// TIA Portal V18 export
FUNCTION "Recirculation Sequences" : Void   // FC12, LAD
{ S7_Optimized_Access := 'TRUE' }
VERSION : 0.1
// stored: AutoNumber true, IsIECCheckEnabled false, SetENOAutomatically false, UDAEnableTagReadback false
   VAR_TEMP   // added for the SCL form of the ladder/FBD networks
      _w1 : Bool;
   END_VAR
BEGIN

REGION Network 1: A selection
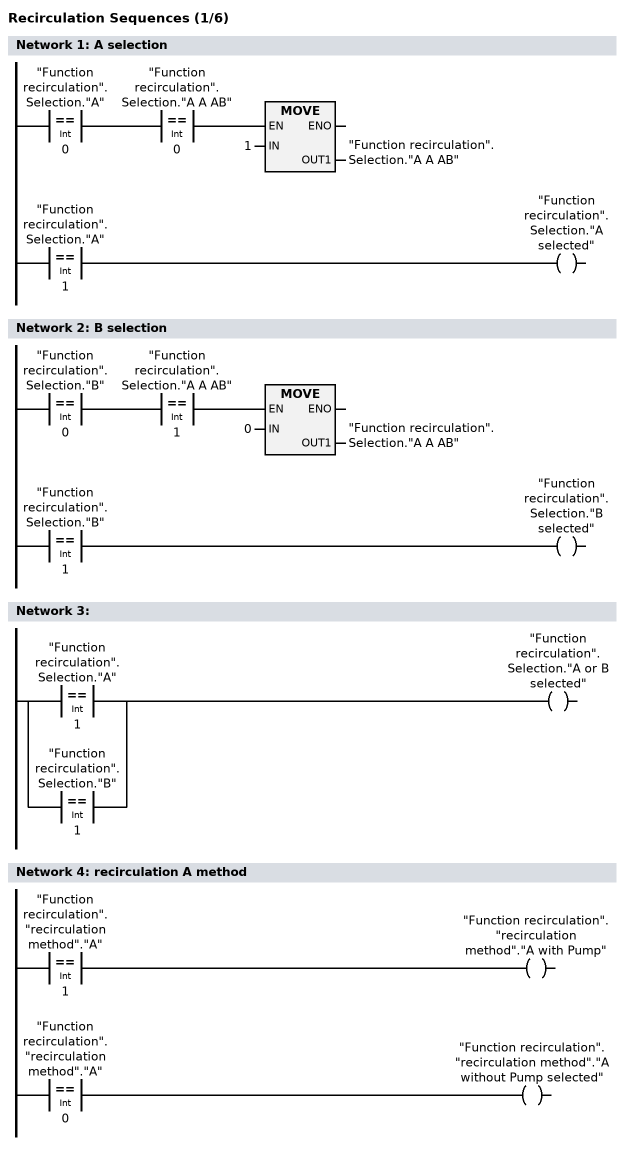
   RUNG wire#powerrail
      { S7_Templates := "SrcType := Int" } EQ_Contact(in1 := "Function recirculation".Selection."A", in2 := 0)
      { S7_Templates := "SrcType := Int" } EQ_Contact(in1 := "Function recirculation".Selection."A A AB", in2 := 0)
      Move(in := 1, out1 => "Function recirculation".Selection."A A AB")
   END_RUNG
   RUNG wire#powerrail
      { S7_Templates := "SrcType := Int" } EQ_Contact(in1 := "Function recirculation".Selection."A", in2 := 1)
      Coil( "Function recirculation".Selection."A selected" )
   END_RUNG
   // the same network as SCL:
   IF ("Function recirculation".Selection."A" = 0) AND ("Function recirculation".Selection."A A AB" = 0) THEN
       "Function recirculation".Selection."A A AB" := 1;
   END_IF;
   "Function recirculation".Selection."A selected" := "Function recirculation".Selection."A" = 1;
END_REGION

REGION Network 2: B selection
   RUNG wire#powerrail
      { S7_Templates := "SrcType := Int" } EQ_Contact(in1 := "Function recirculation".Selection."B", in2 := 0)
      { S7_Templates := "SrcType := Int" } EQ_Contact(in1 := "Function recirculation".Selection."A A AB", in2 := 1)
      Move(in := 0, out1 => "Function recirculation".Selection."A A AB")
   END_RUNG
   RUNG wire#powerrail
      { S7_Templates := "SrcType := Int" } EQ_Contact(in1 := "Function recirculation".Selection."B", in2 := 1)
      Coil( "Function recirculation".Selection."B selected" )
   END_RUNG
   // the same network as SCL:
   IF ("Function recirculation".Selection."B" = 0) AND ("Function recirculation".Selection."A A AB" = 1) THEN
       "Function recirculation".Selection."A A AB" := 0;
   END_IF;
   "Function recirculation".Selection."B selected" := "Function recirculation".Selection."B" = 1;
END_REGION

REGION Network 3
   RUNG wire#powerrail
      { S7_Templates := "SrcType := Int" } EQ_Contact(in1 := "Function recirculation".Selection."A", in2 := 1)
      wire#w1
      Coil( "Function recirculation".Selection."A or B selected" )
   END_RUNG
   RUNG wire#powerrail
      { S7_Templates := "SrcType := Int" } EQ_Contact(in1 := "Function recirculation".Selection."B", in2 := 1)
   END_RUNG wire#w1
   // the same network as SCL:
   "Function recirculation".Selection."A or B selected" := ("Function recirculation".Selection."A" = 1) OR ("Function recirculation".Selection."B" = 1);
END_REGION

REGION Network 4: recirculation A method
   RUNG wire#powerrail
      { S7_Templates := "SrcType := Int" } EQ_Contact(in1 := "Function recirculation"."recirculation method"."A", in2 := 1)
      Coil( "Function recirculation"."recirculation method"."A with Pump" )
   END_RUNG
   RUNG wire#powerrail
      { S7_Templates := "SrcType := Int" } EQ_Contact(in1 := "Function recirculation"."recirculation method"."A", in2 := 0)
      Coil( "Function recirculation"."recirculation method"."A without Pump selected" )
   END_RUNG
   // the same network as SCL:
   "Function recirculation"."recirculation method"."A with Pump" := "Function recirculation"."recirculation method"."A" = 1;
   "Function recirculation"."recirculation method"."A without Pump selected" := "Function recirculation"."recirculation method"."A" = 0;
END_REGION

REGION Network 5: recirculation B method
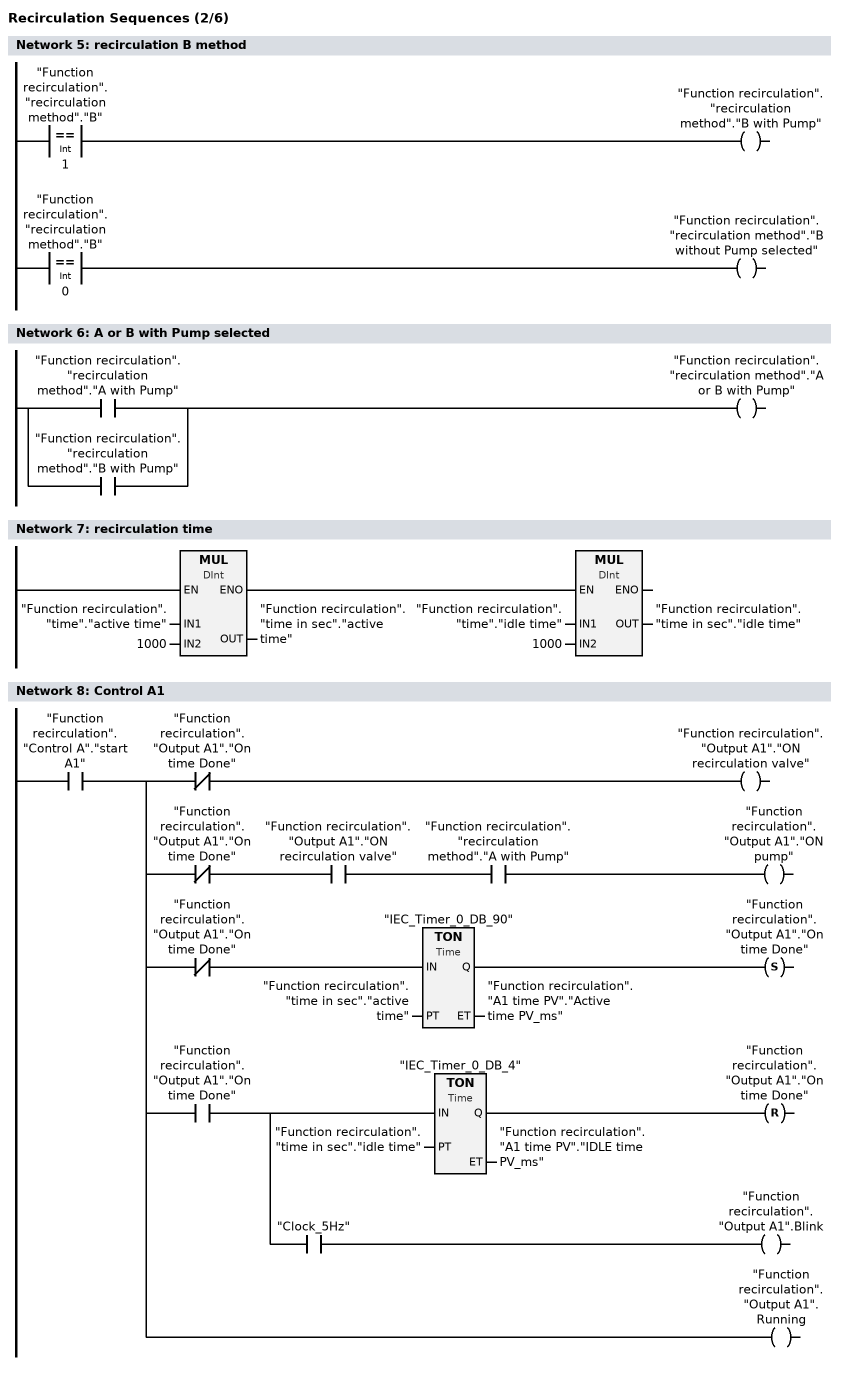
   RUNG wire#powerrail
      { S7_Templates := "SrcType := Int" } EQ_Contact(in1 := "Function recirculation"."recirculation method"."B", in2 := 1)
      Coil( "Function recirculation"."recirculation method"."B with Pump" )
   END_RUNG
   RUNG wire#powerrail
      { S7_Templates := "SrcType := Int" } EQ_Contact(in1 := "Function recirculation"."recirculation method"."B", in2 := 0)
      Coil( "Function recirculation"."recirculation method"."B without Pump selected" )
   END_RUNG
   // the same network as SCL:
   "Function recirculation"."recirculation method"."B with Pump" := "Function recirculation"."recirculation method"."B" = 1;
   "Function recirculation"."recirculation method"."B without Pump selected" := "Function recirculation"."recirculation method"."B" = 0;
END_REGION

REGION Network 6: A or B with Pump selected
   RUNG wire#powerrail
      Contact( "Function recirculation"."recirculation method"."A with Pump" )
      wire#w1
      Coil( "Function recirculation"."recirculation method"."A or B with Pump" )
   END_RUNG
   RUNG wire#powerrail
      Contact( "Function recirculation"."recirculation method"."B with Pump" )
   END_RUNG wire#w1
   // the same network as SCL:
   "Function recirculation"."recirculation method"."A or B with Pump" := "Function recirculation"."recirculation method"."A with Pump" OR "Function recirculation"."recirculation method"."B with Pump";
END_REGION

REGION Network 7: recirculation time
   RUNG wire#powerrail
      { S7_Templates := "SrcType := DInt" } Mul(in1 := "Function recirculation"."time"."active time", in2 := 1000, out => "Function recirculation"."time in sec"."active time")
      { S7_Templates := "SrcType := DInt" } Mul(in1 := "Function recirculation"."time"."idle time", in2 := 1000, out => "Function recirculation"."time in sec"."idle time")
   END_RUNG
   // the same network as SCL:
   "Function recirculation"."time in sec"."active time" := "Function recirculation"."time"."active time" * 1000;
   "Function recirculation"."time in sec"."idle time" := "Function recirculation"."time"."idle time" * 1000;
END_REGION

REGION Network 8: Control A1
   RUNG wire#powerrail
      Contact( "Function recirculation"."Control A"."start A1" )
      wire#w1
      I_Contact( "Function recirculation"."Output A1"."On time Done" )
      Coil( "Function recirculation"."Output A1"."ON recirculation valve" )
   END_RUNG
   RUNG wire#w1
      I_Contact( "Function recirculation"."Output A1"."On time Done" )
      Contact( "Function recirculation"."Output A1"."ON recirculation valve" )
      Contact( "Function recirculation"."recirculation method"."A with Pump" )
      Coil( "Function recirculation"."Output A1"."ON pump" )
   END_RUNG
   RUNG wire#w1
      I_Contact( "Function recirculation"."Output A1"."On time Done" )
      { S7_Templates := "time_type := Time" } "IEC_Timer_0_DB_90".TON(pt := "Function recirculation"."time in sec"."active time", et => "Function recirculation"."A1 time PV"."Active time PV_ms")
      S_Coil( "Function recirculation"."Output A1"."On time Done" )
   END_RUNG
   RUNG wire#w1
      Contact( "Function recirculation"."Output A1"."On time Done" )
      wire#w2
      { S7_Templates := "time_type := Time" } "IEC_Timer_0_DB_4".TON(pt := "Function recirculation"."time in sec"."idle time", et => "Function recirculation"."A1 time PV"."IDLE time PV_ms")
      R_Coil( "Function recirculation"."Output A1"."On time Done" )
   END_RUNG
   RUNG wire#w2
      Contact( "Clock_5Hz" )
      Coil( "Function recirculation"."Output A1".Blink )
   END_RUNG
   RUNG wire#w1
      Coil( "Function recirculation"."Output A1".Running )
   END_RUNG
   // the same network as SCL:
   "Function recirculation"."Output A1"."ON recirculation valve" := "Function recirculation"."Control A"."start A1" AND NOT "Function recirculation"."Output A1"."On time Done";
   "Function recirculation"."Output A1"."ON pump" := "Function recirculation"."Control A"."start A1" AND NOT "Function recirculation"."Output A1"."On time Done" AND "Function recirculation"."Output A1"."ON recirculation valve" AND "Function recirculation"."recirculation method"."A with Pump";
   "IEC_Timer_0_DB_90".TON(IN := "Function recirculation"."Control A"."start A1" AND NOT "Function recirculation"."Output A1"."On time Done",
                           PT := "Function recirculation"."time in sec"."active time",
                           ET => "Function recirculation"."A1 time PV"."Active time PV_ms");
   IF "IEC_Timer_0_DB_90".Q THEN "Function recirculation"."Output A1"."On time Done" := TRUE; END_IF;
   #_w1 := "Function recirculation"."Control A"."start A1" AND "Function recirculation"."Output A1"."On time Done";
   "IEC_Timer_0_DB_4".TON(IN := #_w1,
                          PT := "Function recirculation"."time in sec"."idle time",
                          ET => "Function recirculation"."A1 time PV"."IDLE time PV_ms");
   IF "IEC_Timer_0_DB_4".Q THEN "Function recirculation"."Output A1"."On time Done" := FALSE; END_IF;
   "Function recirculation"."Output A1".Blink := #_w1 AND "Clock_5Hz";
   "Function recirculation"."Output A1".Running := "Function recirculation"."Control A"."start A1";
END_REGION

REGION Network 9: Control A2
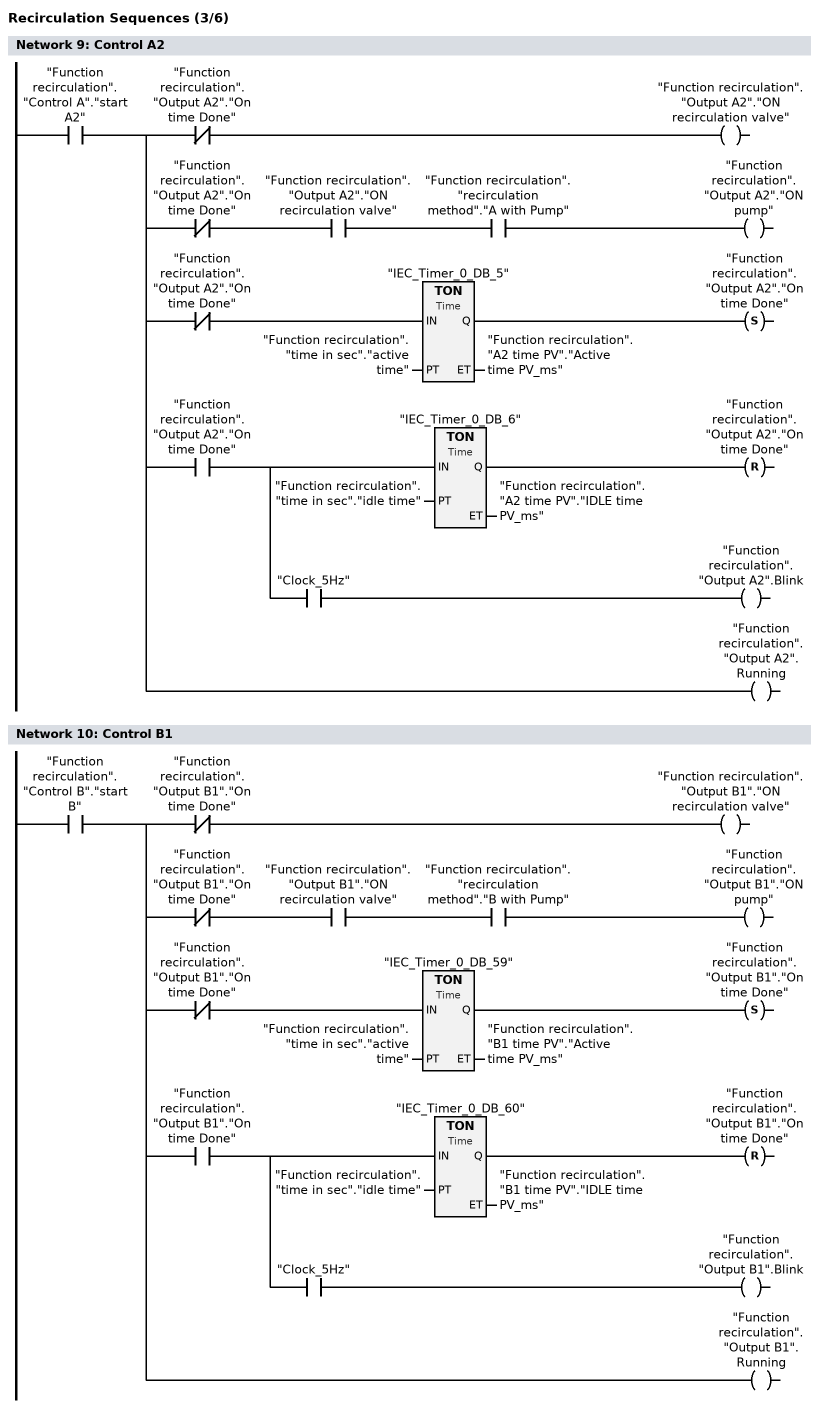
   RUNG wire#powerrail
      Contact( "Function recirculation"."Control A"."start A2" )
      wire#w1
      I_Contact( "Function recirculation"."Output A2"."On time Done" )
      Coil( "Function recirculation"."Output A2"."ON recirculation valve" )
   END_RUNG
   RUNG wire#w1
      I_Contact( "Function recirculation"."Output A2"."On time Done" )
      Contact( "Function recirculation"."Output A2"."ON recirculation valve" )
      Contact( "Function recirculation"."recirculation method"."A with Pump" )
      Coil( "Function recirculation"."Output A2"."ON pump" )
   END_RUNG
   RUNG wire#w1
      I_Contact( "Function recirculation"."Output A2"."On time Done" )
      { S7_Templates := "time_type := Time" } "IEC_Timer_0_DB_5".TON(pt := "Function recirculation"."time in sec"."active time", et => "Function recirculation"."A2 time PV"."Active time PV_ms")
      S_Coil( "Function recirculation"."Output A2"."On time Done" )
   END_RUNG
   RUNG wire#w1
      Contact( "Function recirculation"."Output A2"."On time Done" )
      wire#w2
      { S7_Templates := "time_type := Time" } "IEC_Timer_0_DB_6".TON(pt := "Function recirculation"."time in sec"."idle time", et => "Function recirculation"."A2 time PV"."IDLE time PV_ms")
      R_Coil( "Function recirculation"."Output A2"."On time Done" )
   END_RUNG
   RUNG wire#w2
      Contact( "Clock_5Hz" )
      Coil( "Function recirculation"."Output A2".Blink )
   END_RUNG
   RUNG wire#w1
      Coil( "Function recirculation"."Output A2".Running )
   END_RUNG
   // the same network as SCL:
   "Function recirculation"."Output A2"."ON recirculation valve" := "Function recirculation"."Control A"."start A2" AND NOT "Function recirculation"."Output A2"."On time Done";
   "Function recirculation"."Output A2"."ON pump" := "Function recirculation"."Control A"."start A2" AND NOT "Function recirculation"."Output A2"."On time Done" AND "Function recirculation"."Output A2"."ON recirculation valve" AND "Function recirculation"."recirculation method"."A with Pump";
   "IEC_Timer_0_DB_5".TON(IN := "Function recirculation"."Control A"."start A2" AND NOT "Function recirculation"."Output A2"."On time Done",
                          PT := "Function recirculation"."time in sec"."active time",
                          ET => "Function recirculation"."A2 time PV"."Active time PV_ms");
   IF "IEC_Timer_0_DB_5".Q THEN "Function recirculation"."Output A2"."On time Done" := TRUE; END_IF;
   #_w1 := "Function recirculation"."Control A"."start A2" AND "Function recirculation"."Output A2"."On time Done";
   "IEC_Timer_0_DB_6".TON(IN := #_w1,
                          PT := "Function recirculation"."time in sec"."idle time",
                          ET => "Function recirculation"."A2 time PV"."IDLE time PV_ms");
   IF "IEC_Timer_0_DB_6".Q THEN "Function recirculation"."Output A2"."On time Done" := FALSE; END_IF;
   "Function recirculation"."Output A2".Blink := #_w1 AND "Clock_5Hz";
   "Function recirculation"."Output A2".Running := "Function recirculation"."Control A"."start A2";
END_REGION

REGION Network 10: Control B1
   RUNG wire#powerrail
      Contact( "Function recirculation"."Control B"."start B" )
      wire#w1
      I_Contact( "Function recirculation"."Output B1"."On time Done" )
      Coil( "Function recirculation"."Output B1"."ON recirculation valve" )
   END_RUNG
   RUNG wire#w1
      I_Contact( "Function recirculation"."Output B1"."On time Done" )
      Contact( "Function recirculation"."Output B1"."ON recirculation valve" )
      Contact( "Function recirculation"."recirculation method"."B with Pump" )
      Coil( "Function recirculation"."Output B1"."ON pump" )
   END_RUNG
   RUNG wire#w1
      I_Contact( "Function recirculation"."Output B1"."On time Done" )
      { S7_Templates := "time_type := Time" } "IEC_Timer_0_DB_59".TON(pt := "Function recirculation"."time in sec"."active time", et => "Function recirculation"."B1 time PV"."Active time PV_ms")
      S_Coil( "Function recirculation"."Output B1"."On time Done" )
   END_RUNG
   RUNG wire#w1
      Contact( "Function recirculation"."Output B1"."On time Done" )
      wire#w2
      { S7_Templates := "time_type := Time" } "IEC_Timer_0_DB_60".TON(pt := "Function recirculation"."time in sec"."idle time", et => "Function recirculation"."B1 time PV"."IDLE time PV_ms")
      R_Coil( "Function recirculation"."Output B1"."On time Done" )
   END_RUNG
   RUNG wire#w2
      Contact( "Clock_5Hz" )
      Coil( "Function recirculation"."Output B1".Blink )
   END_RUNG
   RUNG wire#w1
      Coil( "Function recirculation"."Output B1".Running )
   END_RUNG
   // the same network as SCL:
   "Function recirculation"."Output B1"."ON recirculation valve" := "Function recirculation"."Control B"."start B" AND NOT "Function recirculation"."Output B1"."On time Done";
   "Function recirculation"."Output B1"."ON pump" := "Function recirculation"."Control B"."start B" AND NOT "Function recirculation"."Output B1"."On time Done" AND "Function recirculation"."Output B1"."ON recirculation valve" AND "Function recirculation"."recirculation method"."B with Pump";
   "IEC_Timer_0_DB_59".TON(IN := "Function recirculation"."Control B"."start B" AND NOT "Function recirculation"."Output B1"."On time Done",
                           PT := "Function recirculation"."time in sec"."active time",
                           ET => "Function recirculation"."B1 time PV"."Active time PV_ms");
   IF "IEC_Timer_0_DB_59".Q THEN "Function recirculation"."Output B1"."On time Done" := TRUE; END_IF;
   #_w1 := "Function recirculation"."Control B"."start B" AND "Function recirculation"."Output B1"."On time Done";
   "IEC_Timer_0_DB_60".TON(IN := #_w1,
                           PT := "Function recirculation"."time in sec"."idle time",
                           ET => "Function recirculation"."B1 time PV"."IDLE time PV_ms");
   IF "IEC_Timer_0_DB_60".Q THEN "Function recirculation"."Output B1"."On time Done" := FALSE; END_IF;
   "Function recirculation"."Output B1".Blink := #_w1 AND "Clock_5Hz";
   "Function recirculation"."Output B1".Running := "Function recirculation"."Control B"."start B";
END_REGION

REGION Network 11: Recirculation A Active time PV
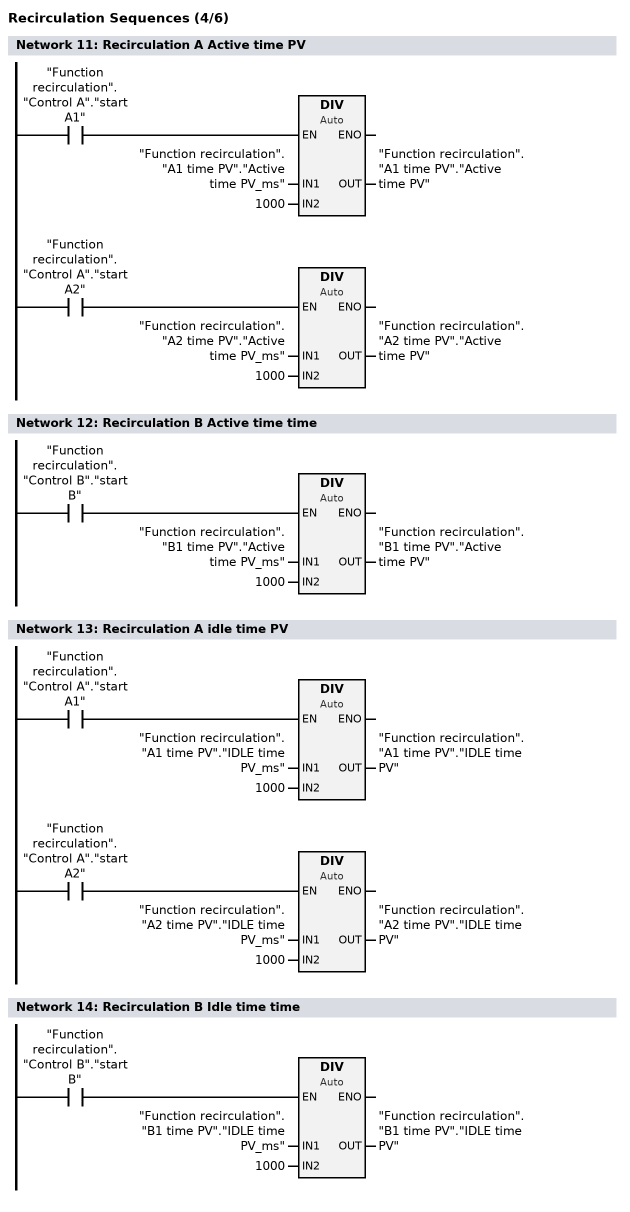
   RUNG wire#powerrail
      Contact( "Function recirculation"."Control A"."start A1" )
      Div(in1 := "Function recirculation"."A1 time PV"."Active time PV_ms", in2 := 1000, out => "Function recirculation"."A1 time PV"."Active time PV")
   END_RUNG
   RUNG wire#powerrail
      Contact( "Function recirculation"."Control A"."start A2" )
      Div(in1 := "Function recirculation"."A2 time PV"."Active time PV_ms", in2 := 1000, out => "Function recirculation"."A2 time PV"."Active time PV")
   END_RUNG
   // the same network as SCL:
   IF "Function recirculation"."Control A"."start A1" THEN
       "Function recirculation"."A1 time PV"."Active time PV" := "Function recirculation"."A1 time PV"."Active time PV_ms" / 1000;
   END_IF;
   IF "Function recirculation"."Control A"."start A2" THEN
       "Function recirculation"."A2 time PV"."Active time PV" := "Function recirculation"."A2 time PV"."Active time PV_ms" / 1000;
   END_IF;
END_REGION

REGION Network 12: Recirculation B Active time time
   RUNG wire#powerrail
      Contact( "Function recirculation"."Control B"."start B" )
      Div(in1 := "Function recirculation"."B1 time PV"."Active time PV_ms", in2 := 1000, out => "Function recirculation"."B1 time PV"."Active time PV")
   END_RUNG
   // the same network as SCL:
   IF "Function recirculation"."Control B"."start B" THEN
       "Function recirculation"."B1 time PV"."Active time PV" := "Function recirculation"."B1 time PV"."Active time PV_ms" / 1000;
   END_IF;
END_REGION

REGION Network 13: Recirculation A idle time PV
   RUNG wire#powerrail
      Contact( "Function recirculation"."Control A"."start A1" )
      Div(in1 := "Function recirculation"."A1 time PV"."IDLE time PV_ms", in2 := 1000, out => "Function recirculation"."A1 time PV"."IDLE time PV")
   END_RUNG
   RUNG wire#powerrail
      Contact( "Function recirculation"."Control A"."start A2" )
      Div(in1 := "Function recirculation"."A2 time PV"."IDLE time PV_ms", in2 := 1000, out => "Function recirculation"."A2 time PV"."IDLE time PV")
   END_RUNG
   // the same network as SCL:
   IF "Function recirculation"."Control A"."start A1" THEN
       "Function recirculation"."A1 time PV"."IDLE time PV" := "Function recirculation"."A1 time PV"."IDLE time PV_ms" / 1000;
   END_IF;
   IF "Function recirculation"."Control A"."start A2" THEN
       "Function recirculation"."A2 time PV"."IDLE time PV" := "Function recirculation"."A2 time PV"."IDLE time PV_ms" / 1000;
   END_IF;
END_REGION

REGION Network 14: Recirculation B Idle time time
   RUNG wire#powerrail
      Contact( "Function recirculation"."Control B"."start B" )
      Div(in1 := "Function recirculation"."B1 time PV"."IDLE time PV_ms", in2 := 1000, out => "Function recirculation"."B1 time PV"."IDLE time PV")
   END_RUNG
   // the same network as SCL:
   IF "Function recirculation"."Control B"."start B" THEN
       "Function recirculation"."B1 time PV"."IDLE time PV" := "Function recirculation"."B1 time PV"."IDLE time PV_ms" / 1000;
   END_IF;
END_REGION

REGION Network 15: A1 Active time to HMI
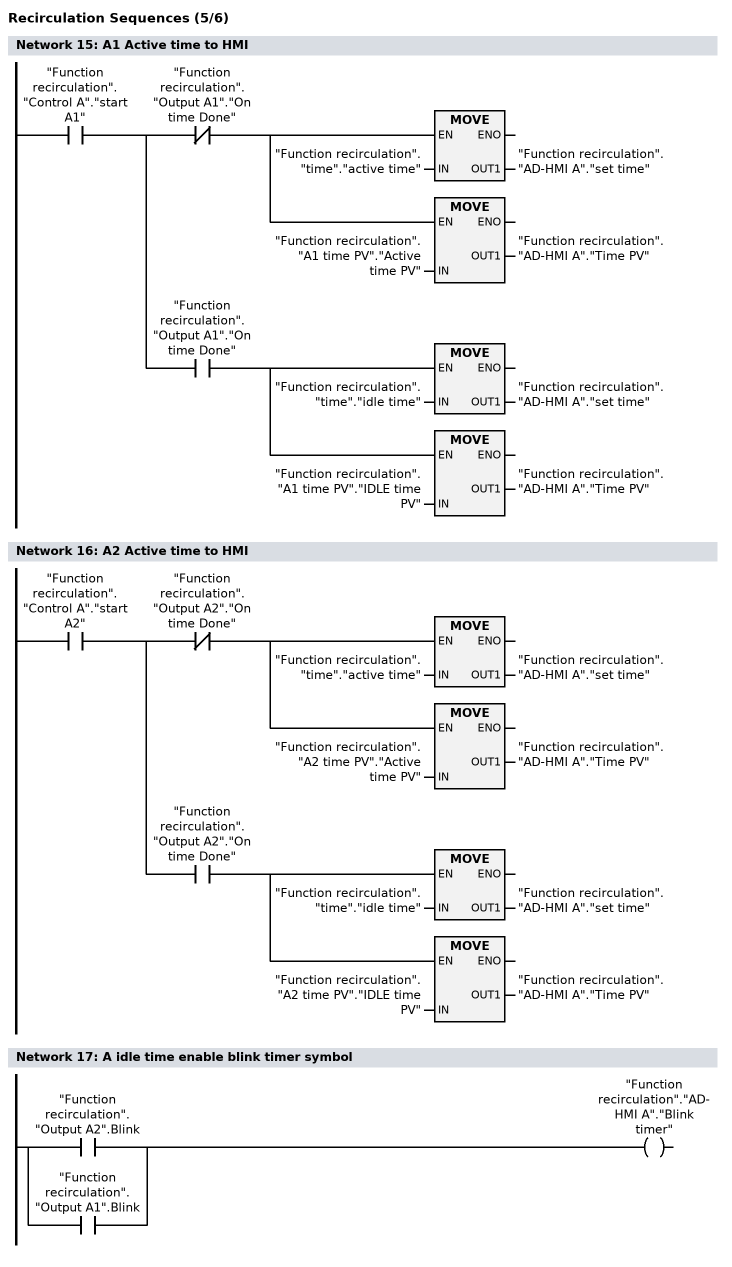
   RUNG wire#powerrail
      Contact( "Function recirculation"."Control A"."start A1" )
      wire#w1
      I_Contact( "Function recirculation"."Output A1"."On time Done" )
      wire#w2
      Move(in := "Function recirculation"."time"."active time", out1 => "Function recirculation"."AD-HMI A"."set time")
   END_RUNG
   RUNG wire#w2
      Move(in := "Function recirculation"."A1 time PV"."Active time PV", out1 => "Function recirculation"."AD-HMI A"."Time PV")
   END_RUNG
   RUNG wire#w1
      Contact( "Function recirculation"."Output A1"."On time Done" )
      wire#w3
      Move(in := "Function recirculation"."time"."idle time", out1 => "Function recirculation"."AD-HMI A"."set time")
   END_RUNG
   RUNG wire#w3
      Move(in := "Function recirculation"."A1 time PV"."IDLE time PV", out1 => "Function recirculation"."AD-HMI A"."Time PV")
   END_RUNG
   // the same network as SCL:
   IF "Function recirculation"."Control A"."start A1" AND NOT "Function recirculation"."Output A1"."On time Done" THEN
       "Function recirculation"."AD-HMI A"."set time" := "Function recirculation"."time"."active time";
       "Function recirculation"."AD-HMI A"."Time PV" := "Function recirculation"."A1 time PV"."Active time PV";
   END_IF;
   IF "Function recirculation"."Control A"."start A1" AND "Function recirculation"."Output A1"."On time Done" THEN
       "Function recirculation"."AD-HMI A"."set time" := "Function recirculation"."time"."idle time";
       "Function recirculation"."AD-HMI A"."Time PV" := "Function recirculation"."A1 time PV"."IDLE time PV";
   END_IF;
END_REGION

REGION Network 16: A2 Active time to HMI
   RUNG wire#powerrail
      Contact( "Function recirculation"."Control A"."start A2" )
      wire#w1
      I_Contact( "Function recirculation"."Output A2"."On time Done" )
      wire#w2
      Move(in := "Function recirculation"."time"."active time", out1 => "Function recirculation"."AD-HMI A"."set time")
   END_RUNG
   RUNG wire#w2
      Move(in := "Function recirculation"."A2 time PV"."Active time PV", out1 => "Function recirculation"."AD-HMI A"."Time PV")
   END_RUNG
   RUNG wire#w1
      Contact( "Function recirculation"."Output A2"."On time Done" )
      wire#w3
      Move(in := "Function recirculation"."time"."idle time", out1 => "Function recirculation"."AD-HMI A"."set time")
   END_RUNG
   RUNG wire#w3
      Move(in := "Function recirculation"."A2 time PV"."IDLE time PV", out1 => "Function recirculation"."AD-HMI A"."Time PV")
   END_RUNG
   // the same network as SCL:
   IF "Function recirculation"."Control A"."start A2" AND NOT "Function recirculation"."Output A2"."On time Done" THEN
       "Function recirculation"."AD-HMI A"."set time" := "Function recirculation"."time"."active time";
       "Function recirculation"."AD-HMI A"."Time PV" := "Function recirculation"."A2 time PV"."Active time PV";
   END_IF;
   IF "Function recirculation"."Control A"."start A2" AND "Function recirculation"."Output A2"."On time Done" THEN
       "Function recirculation"."AD-HMI A"."set time" := "Function recirculation"."time"."idle time";
       "Function recirculation"."AD-HMI A"."Time PV" := "Function recirculation"."A2 time PV"."IDLE time PV";
   END_IF;
END_REGION

REGION Network 17: A idle time enable blink timer symbol
   RUNG wire#powerrail
      Contact( "Function recirculation"."Output A2".Blink )
      wire#w1
      Coil( "Function recirculation"."AD-HMI A"."Blink timer" )
   END_RUNG
   RUNG wire#powerrail
      Contact( "Function recirculation"."Output A1".Blink )
   END_RUNG wire#w1
   // the same network as SCL:
   "Function recirculation"."AD-HMI A"."Blink timer" := "Function recirculation"."Output A2".Blink OR "Function recirculation"."Output A1".Blink;
END_REGION

REGION Network 18: B Active time to HMI
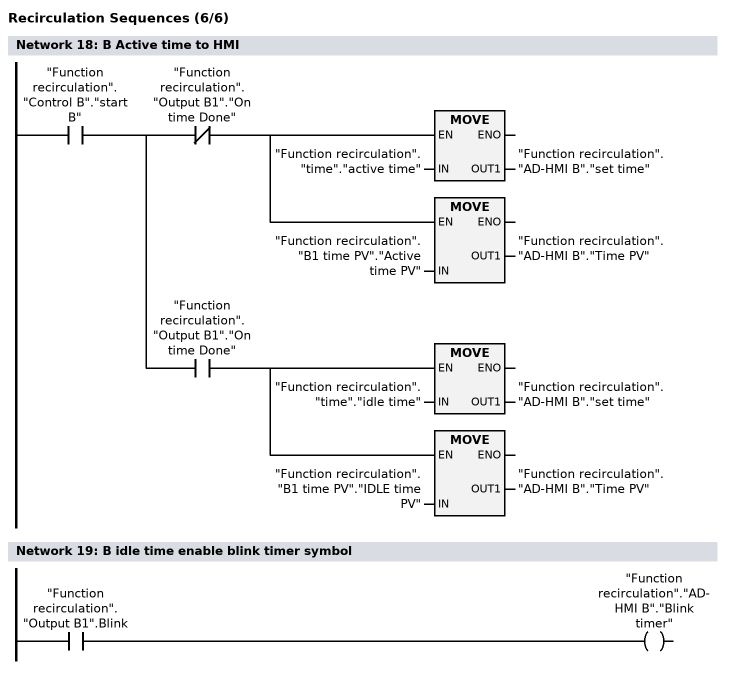
   RUNG wire#powerrail
      Contact( "Function recirculation"."Control B"."start B" )
      wire#w1
      I_Contact( "Function recirculation"."Output B1"."On time Done" )
      wire#w2
      Move(in := "Function recirculation"."time"."active time", out1 => "Function recirculation"."AD-HMI B"."set time")
   END_RUNG
   RUNG wire#w2
      Move(in := "Function recirculation"."B1 time PV"."Active time PV", out1 => "Function recirculation"."AD-HMI B"."Time PV")
   END_RUNG
   RUNG wire#w1
      Contact( "Function recirculation"."Output B1"."On time Done" )
      wire#w3
      Move(in := "Function recirculation"."time"."idle time", out1 => "Function recirculation"."AD-HMI B"."set time")
   END_RUNG
   RUNG wire#w3
      Move(in := "Function recirculation"."B1 time PV"."IDLE time PV", out1 => "Function recirculation"."AD-HMI B"."Time PV")
   END_RUNG
   // the same network as SCL:
   IF "Function recirculation"."Control B"."start B" AND NOT "Function recirculation"."Output B1"."On time Done" THEN
       "Function recirculation"."AD-HMI B"."set time" := "Function recirculation"."time"."active time";
       "Function recirculation"."AD-HMI B"."Time PV" := "Function recirculation"."B1 time PV"."Active time PV";
   END_IF;
   IF "Function recirculation"."Control B"."start B" AND "Function recirculation"."Output B1"."On time Done" THEN
       "Function recirculation"."AD-HMI B"."set time" := "Function recirculation"."time"."idle time";
       "Function recirculation"."AD-HMI B"."Time PV" := "Function recirculation"."B1 time PV"."IDLE time PV";
   END_IF;
END_REGION

REGION Network 19: B idle time enable blink timer symbol
   RUNG wire#powerrail
      Contact( "Function recirculation"."Output B1".Blink )
      Coil( "Function recirculation"."AD-HMI B"."Blink timer" )
   END_RUNG
   // the same network as SCL:
   "Function recirculation"."AD-HMI B"."Blink timer" := "Function recirculation"."Output B1".Blink;
END_REGION
END_FUNCTION
